                                        FB_Bacnet.StartStopCommand_142.bEnWrite := TRUE;
                                        FB_Bacnet.StartStopCommand_142.bVal := FALSE;
                                    16: 
                                        
                                        FB_Bacnet.StartStopCommand_143.bEnWrite := TRUE;
                                        FB_Bacnet.StartStopCommand_143.bVal := FALSE;
                                    17: 
                                        
                                        FB_Bacnet.StartStopCommand_144.bEnWrite := TRUE;
                                        FB_Bacnet.StartStopCommand_144.bVal := FALSE;
                                    18: 
                                        
                                        FB_Bacnet.StartStopCommand_145.bEnWrite := TRUE;
                                        FB_Bacnet.StartStopCommand_145.bVal := FALSE;
                                    19: 
                                        
                                        FB_Bacnet.StartStopCommand_146.bEnWrite := TRUE;
                                        FB_Bacnet.StartStopCommand_146.bVal := FALSE;
                                    20: 
                                        
                                        FB_Bacnet.StartStopCommand_147.bEnWrite := TRUE;
                                        FB_Bacnet.StartStopCommand_147.bVal := FALSE;
                                    21: 
                                        
                                        FB_Bacnet.StartStopCommand_148.bEnWrite := TRUE;
                                        FB_Bacnet.StartStopCommand_148.bVal := FALSE;
                                    22: 
                                        
                                        FB_Bacnet.StartStopCommand_176.bEnWrite := TRUE;
                                        FB_Bacnet.StartStopCommand_176.bVal := FALSE;
                                    23: 
                                        
                                        FB_Bacnet_b.StartStopCommand_241.bEnWrite := TRUE;
                                        FB_Bacnet_b.StartStopCommand_241.bVal := FALSE;
                                    24: 
                                        
                                        FB_Bacnet_b.StartStopCommand_227.bEnWrite := TRUE;
                                        FB_Bacnet_b.StartStopCommand_227.bVal := FALSE;
                                END_CASE
                            END_IF
                        END_FOR
                    END_IF
                END_IF
            END_IF

            // Weekend schedule
            IF currD = 0 OR currD = 6 THEN
                IF (wSchedWEHourStartF7_ <> wSchedWEHourEndF7_ OR wSchedWEMinStartF7_ <> wSchedWEMinEndF7_) THEN
                    // Schedule Unit ON
                    IF wSchedWEHourStartF7_ = currH AND wSchedWEMinStartF7_ = currM AND NOT bUnitTriggered THEN
                        bUnitTriggered := TRUE;
                        FOR i := 1 TO 24 DO
                            // Send command unit ON
                            IF bUnitF7_[i] THEN 
                                CASE i OF
                                    1: 
                                        
                                        FB_Bacnet.StartStopCommand_128.bEnWrite := TRUE;
                                        FB_Bacnet.StartStopCommand_128.bVal := TRUE;
                                    2: 
                                        
                                        FB_Bacnet.StartStopCommand_129.bEnWrite := TRUE;
                                        FB_Bacnet.StartStopCommand_129.bVal := TRUE;
                                    3: 
                                        
                                        FB_Bacnet.StartStopCommand_130.bEnWrite := TRUE;
                                        FB_Bacnet.StartStopCommand_130.bVal := TRUE;
                                    4: 
                                        
                                        FB_Bacnet.StartStopCommand_131.bEnWrite := TRUE;
                                        FB_Bacnet.StartStopCommand_131.bVal := TRUE;
                                    5: 
                                        
                                        FB_Bacnet.StartStopCommand_132.bEnWrite := TRUE;
                                        FB_Bacnet.StartStopCommand_132.bVal := TRUE;
                                    6: 
                                        
                                        FB_Bacnet.StartStopCommand_133.bEnWrite := TRUE;
                                        FB_Bacnet.StartStopCommand_133.bVal := TRUE;
                                    7: 
                                        
                                        FB_Bacnet.StartStopCommand_134.bEnWrite := TRUE;
                                        FB_Bacnet.StartStopCommand_134.bVal := TRUE;
                                    8: 
                                        
                                        FB_Bacnet.StartStopCommand_135.bEnWrite := TRUE;
                                        FB_Bacnet.StartStopCommand_135.bVal := TRUE;
                                    9: 
                                        
                                        FB_Bacnet.StartStopCommand_136.bEnWrite := TRUE;
                                        FB_Bacnet.StartStopCommand_136.bVal := TRUE;
                                    10: 
                                        
                                        FB_Bacnet.StartStopCommand_137.bEnWrite := TRUE;
                                        FB_Bacnet.StartStopCommand_137.bVal := TRUE;
                                    11: 
                                        
                                        FB_Bacnet.StartStopCommand_138.bEnWrite := TRUE;
                                        FB_Bacnet.StartStopCommand_138.bVal := TRUE;
                                    12: 
                                        
                                        FB_Bacnet.StartStopCommand_139.bEnWrite := TRUE;
                                        FB_Bacnet.StartStopCommand_139.bVal := TRUE;
                                    13: 
                                        
                                        FB_Bacnet.StartStopCommand_140.bEnWrite := TRUE;
                                        FB_Bacnet.StartStopCommand_140.bVal := TRUE;
                                    14: 
                                        
                                        FB_Bacnet.StartStopCommand_141.bEnWrite := TRUE;
                                        FB_Bacnet.StartStopCommand_141.bVal := TRUE;
                                    15: 
                                        
                                        FB_Bacnet.StartStopCommand_142.bEnWrite := TRUE;
                                        FB_Bacnet.StartStopCommand_142.bVal := TRUE;
                                    16: 
                                        
                                        FB_Bacnet.StartStopCommand_143.bEnWrite := TRUE;
                                        FB_Bacnet.StartStopCommand_143.bVal := TRUE;
                                    17: 
                                        
                                        FB_Bacnet.StartStopCommand_144.bEnWrite := TRUE;
                                        FB_Bacnet.StartStopCommand_144.bVal := TRUE;
                                    18: 
                                        
                                        FB_Bacnet.StartStopCommand_145.bEnWrite := TRUE;
                                        FB_Bacnet.StartStopCommand_145.bVal := TRUE;
                                    19: 
                                        
                                        FB_Bacnet.StartStopCommand_146.bEnWrite := TRUE;
                                        FB_Bacnet.StartStopCommand_146.bVal := TRUE;
                                    20: 
                                        
                                        FB_Bacnet.StartStopCommand_147.bEnWrite := TRUE;
                                        FB_Bacnet.StartStopCommand_147.bVal := TRUE;
                                    21: 
                                        
                                        FB_Bacnet.StartStopCommand_148.bEnWrite := TRUE;
                                        FB_Bacnet.StartStopCommand_148.bVal := TRUE;
                                    22: 
                                        
                                        FB_Bacnet.StartStopCommand_176.bEnWrite := TRUE;
                                        FB_Bacnet.StartStopCommand_176.bVal := TRUE;
                                    23: 
                                        
                                        FB_Bacnet_b.StartStopCommand_241.bEnWrite := TRUE;
                                        FB_Bacnet_b.StartStopCommand_241.bVal := TRUE;
                                    24: 
                                        
                                        FB_Bacnet_b.StartStopCommand_227.bEnWrite := TRUE;
                                        FB_Bacnet_b.StartStopCommand_227.bVal := TRUE;
                                END_CASE
                            END_IF
                        END_FOR
                    END_IF
                    // Schedule Unit OFF
                    IF wSchedWEHourEndF7_ = currH AND wSchedWEMinEndF7_ = currM AND NOT bUnitTriggered THEN
                        bUnitTriggered := TRUE;
                        FOR i := 1 TO 24 DO
                            // Send command unit OFF
                            IF bUnitF7_[i] THEN 
                                CASE i OF
                                    1: 
                                        
                                        FB_Bacnet.StartStopCommand_128.bEnWrite := TRUE;
                                        FB_Bacnet.StartStopCommand_128.bVal := FALSE;
                                    2: 
                                        
                                        FB_Bacnet.StartStopCommand_129.bEnWrite := TRUE;
                                        FB_Bacnet.StartStopCommand_129.bVal := FALSE;
                                    3: 
                                        
                                        FB_Bacnet.StartStopCommand_130.bEnWrite := TRUE;
                                        FB_Bacnet.StartStopCommand_130.bVal := FALSE;
                                    4: 
                                        
                                        FB_Bacnet.StartStopCommand_131.bEnWrite := TRUE;
                                        FB_Bacnet.StartStopCommand_131.bVal := FALSE;
                                    5: 
                                        
                                        FB_Bacnet.StartStopCommand_132.bEnWrite := TRUE;
                                        FB_Bacnet.StartStopCommand_132.bVal := FALSE;
                                    6: 
                                        
                                        FB_Bacnet.StartStopCommand_133.bEnWrite := TRUE;
                                        FB_Bacnet.StartStopCommand_133.bVal := FALSE;
                                    7: 
                                        
                                        FB_Bacnet.StartStopCommand_134.bEnWrite := TRUE;
                                        FB_Bacnet.StartStopCommand_134.bVal := FALSE;
                                    8: 
                                        
                                        FB_Bacnet.StartStopCommand_135.bEnWrite := TRUE;
                                        FB_Bacnet.StartStopCommand_135.bVal := FALSE;
                                    9: 
                                        
                                        FB_Bacnet.StartStopCommand_136.bEnWrite := TRUE;
                                        FB_Bacnet.StartStopCommand_136.bVal := FALSE;
                                    10: 
                                        
                                        FB_Bacnet.StartStopCommand_137.bEnWrite := TRUE;
                                        FB_Bacnet.StartStopCommand_137.bVal := FALSE;
                                    11: 
                                        
                                        FB_Bacnet.StartStopCommand_138.bEnWrite := TRUE;
                                        FB_Bacnet.StartStopCommand_138.bVal := FALSE;
                                    12: 
                                        
                                        FB_Bacnet.StartStopCommand_139.bEnWrite := TRUE;
                                        FB_Bacnet.StartStopCommand_139.bVal := FALSE;
                                    13: 
                                        
                                        FB_Bacnet.StartStopCommand_140.bEnWrite := TRUE;
                                        FB_Bacnet.StartStopCommand_140.bVal := FALSE;
                                    14: 
                                        
                                        FB_Bacnet.StartStopCommand_141.bEnWrite := TRUE;
                                        FB_Bacnet.StartStopCommand_141.bVal := FALSE;
                                    15: 
                                        
                                        FB_Bacnet.StartStopCommand_142.bEnWrite := TRUE;
                                        FB_Bacnet.StartStopCommand_142.bVal := FALSE;
                                    16: 
                                        
                                        FB_Bacnet.StartStopCommand_143.bEnWrite := TRUE;
                                        FB_Bacnet.StartStopCommand_143.bVal := FALSE;
                                    17: 
                                        
                                        FB_Bacnet.StartStopCommand_144.bEnWrite := TRUE;
                                        FB_Bacnet.StartStopCommand_144.bVal := FALSE;
                                    18: 
                                        
                                        FB_Bacnet.StartStopCommand_145.bEnWrite := TRUE;
                                        FB_Bacnet.StartStopCommand_145.bVal := FALSE;
                                    19: 
                                        
                                        FB_Bacnet.StartStopCommand_146.bEnWrite := TRUE;
                                        FB_Bacnet.StartStopCommand_146.bVal := FALSE;
                                    20: 
                                        
                                        FB_Bacnet.StartStopCommand_147.bEnWrite := TRUE;
                                        FB_Bacnet.StartStopCommand_147.bVal := FALSE;
                                    21: 
                                        
                                        FB_Bacnet.StartStopCommand_148.bEnWrite := TRUE;
                                        FB_Bacnet.StartStopCommand_148.bVal := FALSE;
                                    22: 
                                        
                                        FB_Bacnet.StartStopCommand_176.bEnWrite := TRUE;
                                        FB_Bacnet.StartStopCommand_176.bVal := FALSE;
                                    23: 
                                        
                                        FB_Bacnet_b.StartStopCommand_241.bEnWrite := TRUE;
                                        FB_Bacnet_b.StartStopCommand_241.bVal := FALSE;
                                    24: 
                                        
                                        FB_Bacnet_b.StartStopCommand_227.bEnWrite := TRUE;
                                        FB_Bacnet_b.StartStopCommand_227.bVal := FALSE;
                                END_CASE
                            END_IF
                        END_FOR
                    END_IF
                END_IF
            END_IF
        END_IF

END_FUNCTION_BLOCK

// ---- POUs/FB_Scheduler/FB_Scheduler_F8.TcPOU

      FUNCTION_BLOCK FB_Scheduler_F8
      VAR_INPUT
          currH : WORD;
          currM : WORD;
          currD : WORD;
      END_VAR
      VAR_IN_OUT
          FB_Bacnet : FB_BACnet_DAIKIN_MasterStation_III_No_2;
      END_VAR
      VAR
          i : INT;
          bUnitTriggered : BOOL := FALSE; // Flag to track execution
          prevMinute : WORD := 0;        // Track previous minute
      END_VAR
      VAR PERSISTENT
          // Scheduler variables
          bEnSchedF8_ : BOOL := FALSE;
          wSchedWDHourStartF8_, wSchedWDMinStartF8_ : WORD;
          wSchedWEHourStartF8_, wSchedWEMinStartF8_ : WORD;
          wSchedWDHourEndF8_, wSchedWDMinEndF8_ : WORD;
          wSchedWEHourEndF8_, wSchedWEMinEndF8_ : WORD;
          // Unit variables
          bUnitF8_ : ARRAY [1..22] OF BOOL;
      END_VAR


        // Reset trigger flag at minute change or at the exact scheduled time
        IF currM <> prevMinute OR 
           (currH = wSchedWDHourStartF8_ AND currM = wSchedWDMinStartF8_) OR 
           (currH = wSchedWDHourEndF8_ AND currM = wSchedWDMinEndF8_) THEN
            bUnitTriggered := FALSE;
            prevMinute := currM;
        END_IF

        // Unit Schedule Enable
        IF bEnSchedF8_ THEN
            // Weekday schedule
            IF currD >= 1 AND currD <= 5 THEN
                IF (wSchedWDHourStartF8_ <> wSchedWDHourEndF8_ OR wSchedWDMinStartF8_ <> wSchedWDMinEndF8_) THEN
                    // Schedule Unit ON
                    IF wSchedWDHourStartF8_ = currH AND wSchedWDMinStartF8_ = currM AND NOT bUnitTriggered THEN
                        bUnitTriggered := TRUE;
                        FOR i := 1 TO 22 DO
                            // Send command unit ON
                            IF bUnitF8_[i] THEN 
                                CASE i OF
                                    1: 
                                        FB_Bacnet.StartStopCommand_192.bEnWrite := TRUE;
                                        FB_Bacnet.StartStopCommand_192.bVal := TRUE;
                                    2: 
                                        FB_Bacnet.StartStopCommand_193.bEnWrite := TRUE;
                                        FB_Bacnet.StartStopCommand_193.bVal := TRUE;
                                    3: 
                                        FB_Bacnet.StartStopCommand_194.bEnWrite := TRUE;
                                        FB_Bacnet.StartStopCommand_194.bVal := TRUE;
                                    4: 
                                        FB_Bacnet.StartStopCommand_195.bEnWrite := TRUE;
                                        FB_Bacnet.StartStopCommand_195.bVal := TRUE;
                                    5: 
                                        FB_Bacnet.StartStopCommand_196.bEnWrite := TRUE;
                                        FB_Bacnet.StartStopCommand_196.bVal := TRUE;
                                    6: 
                                        FB_Bacnet.StartStopCommand_197.bEnWrite := TRUE;
                                        FB_Bacnet.StartStopCommand_197.bVal := TRUE;
                                    7: 
                                        FB_Bacnet.StartStopCommand_198.bEnWrite := TRUE;
                                        FB_Bacnet.StartStopCommand_198.bVal := TRUE;
                                    8: 
                                        FB_Bacnet.StartStopCommand_199.bEnWrite := TRUE;
                                        FB_Bacnet.StartStopCommand_199.bVal := TRUE;
                                    9: 
                                        FB_Bacnet.StartStopCommand_200.bEnWrite := TRUE;
                                        FB_Bacnet.StartStopCommand_200.bVal := TRUE;
                                    10: 
                                        FB_Bacnet.StartStopCommand_201.bEnWrite := TRUE;
                                        FB_Bacnet.StartStopCommand_201.bVal := TRUE;
                                    11: 
                                        FB_Bacnet.StartStopCommand_202.bEnWrite := TRUE;
                                        FB_Bacnet.StartStopCommand_202.bVal := TRUE;
                                    12: 
                                        FB_Bacnet.StartStopCommand_203.bEnWrite := TRUE;
                                        FB_Bacnet.StartStopCommand_203.bVal := TRUE;
                                    13: 
                                        FB_Bacnet.StartStopCommand_204.bEnWrite := TRUE;
                                        FB_Bacnet.StartStopCommand_204.bVal := TRUE;
                                    14: 
                                        FB_Bacnet.StartStopCommand_205.bEnWrite := TRUE;
                                        FB_Bacnet.StartStopCommand_205.bVal := TRUE;
                                    15: 
                                        FB_Bacnet.StartStopCommand_206.bEnWrite := TRUE;
                                        FB_Bacnet.StartStopCommand_206.bVal := TRUE;
                                    16: 
                                        FB_Bacnet.StartStopCommand_207.bEnWrite := TRUE;
                                        FB_Bacnet.StartStopCommand_207.bVal := TRUE;
                                    17: 
                                        FB_Bacnet.StartStopCommand_208.bEnWrite := TRUE;
                                        FB_Bacnet.StartStopCommand_208.bVal := TRUE;
                                    18: 
                                        FB_Bacnet.StartStopCommand_209.bEnWrite := TRUE;
                                        FB_Bacnet.StartStopCommand_209.bVal := TRUE;
                                    19: 
                                        FB_Bacnet.StartStopCommand_210.bEnWrite := TRUE;
                                        FB_Bacnet.StartStopCommand_210.bVal := TRUE;
                                    20: 
                                        FB_Bacnet.StartStopCommand_211.bEnWrite := TRUE;
                                        FB_Bacnet.StartStopCommand_211.bVal := TRUE;
                                    21: 
                                        FB_Bacnet.StartStopCommand_212.bEnWrite := TRUE;
                                        FB_Bacnet.StartStopCommand_212.bVal := TRUE;
                                    22: 
                                        FB_Bacnet.StartStopCommand_224.bEnWrite := TRUE;
                                        FB_Bacnet.StartStopCommand_224.bVal := TRUE;
                                END_CASE
                            END_IF
                        END_FOR
                    END_IF
                    // Schedule Unit OFF
                    IF wSchedWDHourEndF8_ = currH AND wSchedWDMinEndF8_ = currM AND NOT bUnitTriggered THEN
                        bUnitTriggered := TRUE;
                        FOR i := 1 TO 22 DO
                            // Send command unit OFF
                            IF bUnitF8_[i] THEN 
                                CASE i OF
                                    1: 
                                        FB_Bacnet.StartStopCommand_192.bEnWrite := TRUE;
                                        FB_Bacnet.StartStopCommand_192.bVal := FALSE;
                                    2: 
                                        FB_Bacnet.StartStopCommand_193.bEnWrite := TRUE;
                                        FB_Bacnet.StartStopCommand_193.bVal := FALSE;
                                    3: 
                                        FB_Bacnet.StartStopCommand_194.bEnWrite := TRUE;
                                        FB_Bacnet.StartStopCommand_194.bVal := FALSE;
                                    4: 
                                        FB_Bacnet.StartStopCommand_195.bEnWrite := TRUE;
                                        FB_Bacnet.StartStopCommand_195.bVal := FALSE;
                                    5: 
                                        FB_Bacnet.StartStopCommand_196.bEnWrite := TRUE;
                                        FB_Bacnet.StartStopCommand_196.bVal := FALSE;
                                    6: 
                                        FB_Bacnet.StartStopCommand_197.bEnWrite := TRUE;
                                        FB_Bacnet.StartStopCommand_197.bVal := FALSE;
                                    7: 
                                        FB_Bacnet.StartStopCommand_198.bEnWrite := TRUE;
                                        FB_Bacnet.StartStopCommand_198.bVal := FALSE;
                                    8: 
                                        FB_Bacnet.StartStopCommand_199.bEnWrite := TRUE;
                                        FB_Bacnet.StartStopCommand_199.bVal := FALSE;
                                    9: 
                                        FB_Bacnet.StartStopCommand_200.bEnWrite := TRUE;
                                        FB_Bacnet.StartStopCommand_200.bVal := FALSE;
                                    10: 
                                        FB_Bacnet.StartStopCommand_201.bEnWrite := TRUE;
                                        FB_Bacnet.StartStopCommand_201.bVal := FALSE;
                                    11: 
                                        FB_Bacnet.StartStopCommand_202.bEnWrite := TRUE;
                                        FB_Bacnet.StartStopCommand_202.bVal := FALSE;
                                    12: 
                                        FB_Bacnet.StartStopCommand_203.bEnWrite := TRUE;
                                        FB_Bacnet.StartStopCommand_203.bVal := FALSE;
                                    13: 
                                        FB_Bacnet.StartStopCommand_204.bEnWrite := TRUE;
                                        FB_Bacnet.StartStopCommand_204.bVal := FALSE;
                                    14: 
                                        FB_Bacnet.StartStopCommand_205.bEnWrite := TRUE;
                                        FB_Bacnet.StartStopCommand_205.bVal := FALSE;
                                    15: 
                                        FB_Bacnet.StartStopCommand_206.bEnWrite := TRUE;
                                        FB_Bacnet.StartStopCommand_206.bVal := FALSE;
                                    16: 
                                        FB_Bacnet.StartStopCommand_207.bEnWrite := TRUE;
                                        FB_Bacnet.StartStopCommand_207.bVal := FALSE;
                                    17: 
                                        FB_Bacnet.StartStopCommand_208.bEnWrite := TRUE;
                                        FB_Bacnet.StartStopCommand_208.bVal := FALSE;
                                    18: 
                                        FB_Bacnet.StartStopCommand_209.bEnWrite := TRUE;
                                        FB_Bacnet.StartStopCommand_209.bVal := FALSE;
                                    19: 
                                        FB_Bacnet.StartStopCommand_210.bEnWrite := TRUE;
                                        FB_Bacnet.StartStopCommand_210.bVal := FALSE;
                                    20: 
                                        FB_Bacnet.StartStopCommand_211.bEnWrite := TRUE;
                                        FB_Bacnet.StartStopCommand_211.bVal := FALSE;
                                    21: 
                                        FB_Bacnet.StartStopCommand_212.bEnWrite := TRUE;
                                        FB_Bacnet.StartStopCommand_212.bVal := FALSE;
                                    22: 
                                        FB_Bacnet.StartStopCommand_224.bEnWrite := TRUE;
                                        FB_Bacnet.StartStopCommand_224.bVal := FALSE;
                                END_CASE
                            END_IF
                        END_FOR
                    END_IF
                END_IF
            END_IF

            // Weekend schedule
            IF currD = 0 OR currD = 6 THEN
                IF (wSchedWEHourStartF8_ <> wSchedWEHourEndF8_ OR wSchedWEMinStartF8_ <> wSchedWEMinEndF8_) THEN
                    // Schedule Unit ON
                    IF wSchedWEHourStartF8_ = currH AND wSchedWEMinStartF8_ = currM AND NOT bUnitTriggered THEN
                        bUnitTriggered := TRUE;
                        FOR i := 1 TO 22 DO
                            // Send command unit ON
                            IF bUnitF8_[i] THEN 
                                CASE i OF
                                    1: 
                                        FB_Bacnet.StartStopCommand_192.bEnWrite := TRUE;
                                        FB_Bacnet.StartStopCommand_192.bVal := TRUE;
                                    2: 
                                        FB_Bacnet.StartStopCommand_193.bEnWrite := TRUE;
                                        FB_Bacnet.StartStopCommand_193.bVal := TRUE;
                                    3: 
                                        FB_Bacnet.StartStopCommand_194.bEnWrite := TRUE;
                                        FB_Bacnet.StartStopCommand_194.bVal := TRUE;
                                    4: 
                                        FB_Bacnet.StartStopCommand_195.bEnWrite := TRUE;
                                        FB_Bacnet.StartStopCommand_195.bVal := TRUE;
                                    5: 
                                        FB_Bacnet.StartStopCommand_196.bEnWrite := TRUE;
                                        FB_Bacnet.StartStopCommand_196.bVal := TRUE;
                                    6: 
                                        FB_Bacnet.StartStopCommand_197.bEnWrite := TRUE;
                                        FB_Bacnet.StartStopCommand_197.bVal := TRUE;
                                    7: 
                                        FB_Bacnet.StartStopCommand_198.bEnWrite := TRUE;
                                        FB_Bacnet.StartStopCommand_198.bVal := TRUE;
                                    8: 
                                        FB_Bacnet.StartStopCommand_199.bEnWrite := TRUE;
                                        FB_Bacnet.StartStopCommand_199.bVal := TRUE;
                                    9: 
                                        FB_Bacnet.StartStopCommand_200.bEnWrite := TRUE;
                                        FB_Bacnet.StartStopCommand_200.bVal := TRUE;
                                    10: 
                                        FB_Bacnet.StartStopCommand_201.bEnWrite := TRUE;
                                        FB_Bacnet.StartStopCommand_201.bVal := TRUE;
                                    11: 
                                        FB_Bacnet.StartStopCommand_202.bEnWrite := TRUE;
                                        FB_Bacnet.StartStopCommand_202.bVal := TRUE;
                                    12: 
                                        FB_Bacnet.StartStopCommand_203.bEnWrite := TRUE;
                                        FB_Bacnet.StartStopCommand_203.bVal := TRUE;
                                    13: 
                                        FB_Bacnet.StartStopCommand_204.bEnWrite := TRUE;
                                        FB_Bacnet.StartStopCommand_204.bVal := TRUE;
                                    14: 
                                        FB_Bacnet.StartStopCommand_205.bEnWrite := TRUE;
                                        FB_Bacnet.StartStopCommand_205.bVal := TRUE;
                                    15: 
                                        FB_Bacnet.StartStopCommand_206.bEnWrite := TRUE;
                                        FB_Bacnet.StartStopCommand_206.bVal := TRUE;
                                    16: 
                                        FB_Bacnet.StartStopCommand_207.bEnWrite := TRUE;
                                        FB_Bacnet.StartStopCommand_207.bVal := TRUE;
                                    17: 
                                        FB_Bacnet.StartStopCommand_208.bEnWrite := TRUE;
                                        FB_Bacnet.StartStopCommand_208.bVal := TRUE;
                                    18: 
                                        FB_Bacnet.StartStopCommand_209.bEnWrite := TRUE;
                                        FB_Bacnet.StartStopCommand_209.bVal := TRUE;
                                    19: 
                                        FB_Bacnet.StartStopCommand_210.bEnWrite := TRUE;
                                        FB_Bacnet.StartStopCommand_210.bVal := TRUE;
                                    20: 
                                        FB_Bacnet.StartStopCommand_211.bEnWrite := TRUE;
                                        FB_Bacnet.StartStopCommand_211.bVal := TRUE;
                                    21: 
                                        FB_Bacnet.StartStopCommand_212.bEnWrite := TRUE;
                                        FB_Bacnet.StartStopCommand_212.bVal := TRUE;
                                    22: 
                                        FB_Bacnet.StartStopCommand_224.bEnWrite := TRUE;
                                        FB_Bacnet.StartStopCommand_224.bVal := TRUE;
                                END_CASE
                            END_IF
                        END_FOR
                    END_IF
                    // Schedule Unit OFF
                    IF wSchedWEHourEndF8_ = currH AND wSchedWEMinEndF8_ = currM AND NOT bUnitTriggered THEN
                        bUnitTriggered := TRUE;
                        FOR i := 1 TO 22 DO
                            // Send command unit OFF
                            IF bUnitF8_[i] THEN 
                                CASE i OF
                                    1: 
                                        FB_Bacnet.StartStopCommand_192.bEnWrite := TRUE;
                                        FB_Bacnet.StartStopCommand_192.bVal := FALSE;
                                    2: 
                                        FB_Bacnet.StartStopCommand_193.bEnWrite := TRUE;
                                        FB_Bacnet.StartStopCommand_193.bVal := FALSE;
                                    3: 
                                        FB_Bacnet.StartStopCommand_194.bEnWrite := TRUE;
                                        FB_Bacnet.StartStopCommand_194.bVal := FALSE;
                                    4: 
                                        FB_Bacnet.StartStopCommand_195.bEnWrite := TRUE;
                                        FB_Bacnet.StartStopCommand_195.bVal := FALSE;
                                    5: 
                                        FB_Bacnet.StartStopCommand_196.bEnWrite := TRUE;
                                        FB_Bacnet.StartStopCommand_196.bVal := FALSE;
                                    6: 
                                        FB_Bacnet.StartStopCommand_197.bEnWrite := TRUE;
                                        FB_Bacnet.StartStopCommand_197.bVal := FALSE;
                                    7: 
                                        FB_Bacnet.StartStopCommand_198.bEnWrite := TRUE;
                                        FB_Bacnet.StartStopCommand_198.bVal := FALSE;
                                    8: 
                                        FB_Bacnet.StartStopCommand_199.bEnWrite := TRUE;
                                        FB_Bacnet.StartStopCommand_199.bVal := FALSE;
                                    9: 
                                        FB_Bacnet.StartStopCommand_200.bEnWrite := TRUE;
                                        FB_Bacnet.StartStopCommand_200.bVal := FALSE;
                                    10: 
                                        FB_Bacnet.StartStopCommand_201.bEnWrite := TRUE;
                                        FB_Bacnet.StartStopCommand_201.bVal := FALSE;
                                    11: 
                                        FB_Bacnet.StartStopCommand_202.bEnWrite := TRUE;
                                        FB_Bacnet.StartStopCommand_202.bVal := FALSE;
                                    12: 
                                        FB_Bacnet.StartStopCommand_203.bEnWrite := TRUE;
                                        FB_Bacnet.StartStopCommand_203.bVal := FALSE;
                                    13: 
                                        FB_Bacnet.StartStopCommand_204.bEnWrite := TRUE;
                                        FB_Bacnet.StartStopCommand_204.bVal := FALSE;
                                    14: 
                                        FB_Bacnet.StartStopCommand_205.bEnWrite := TRUE;
                                        FB_Bacnet.StartStopCommand_205.bVal := FALSE;
                                    15: 
                                        FB_Bacnet.StartStopCommand_206.bEnWrite := TRUE;
                                        FB_Bacnet.StartStopCommand_206.bVal := FALSE;
                                    16: 
                                        FB_Bacnet.StartStopCommand_207.bEnWrite := TRUE;
                                        FB_Bacnet.StartStopCommand_207.bVal := FALSE;
                                    17: 
                                        FB_Bacnet.StartStopCommand_208.bEnWrite := TRUE;
                                        FB_Bacnet.StartStopCommand_208.bVal := FALSE;
                                    18: 
                                        FB_Bacnet.StartStopCommand_209.bEnWrite := TRUE;
                                        FB_Bacnet.StartStopCommand_209.bVal := FALSE;
                                    19: 
                                        FB_Bacnet.StartStopCommand_210.bEnWrite := TRUE;
                                        FB_Bacnet.StartStopCommand_210.bVal := FALSE;
                                    20: 
                                        FB_Bacnet.StartStopCommand_211.bEnWrite := TRUE;
                                        FB_Bacnet.StartStopCommand_211.bVal := FALSE;
                                    21: 
                                        FB_Bacnet.StartStopCommand_212.bEnWrite := TRUE;
                                        FB_Bacnet.StartStopCommand_212.bVal := FALSE;
                                    22: 
                                        FB_Bacnet.StartStopCommand_224.bEnWrite := TRUE;
                                        FB_Bacnet.StartStopCommand_224.bVal := FALSE;
                                END_CASE
                            END_IF
                        END_FOR
                    END_IF
                END_IF
            END_IF
        END_IF

END_FUNCTION_BLOCK

// ---- POUs/FB_Scheduler/FB_Scheduler_F9.TcPOU

      FUNCTION_BLOCK FB_Scheduler_F9
      VAR_INPUT
          currH : WORD;
          currM : WORD;
          currD : WORD;
      END_VAR
      VAR_IN_OUT
          FB_Bacnet : FB_BACnet_DAIKIN_MasterStation_III_No_3;
          FB_Bacnet_b : FB_BACnet_DAIKIN_MasterStation_III_No_2;
      END_VAR
      VAR
          i : INT;
          bUnitTriggered : BOOL := FALSE; // Flag to track execution
          prevMinute : WORD := 0;        // Track previous minute
      END_VAR
      VAR PERSISTENT
          // Scheduler variables
          bEnSchedF9_ : BOOL := FALSE;
          wSchedWDHourStartF9_, wSchedWDMinStartF9_ : WORD;
          wSchedWEHourStartF9_, wSchedWEMinStartF9_ : WORD;
          wSchedWDHourEndF9_, wSchedWDMinEndF9_ : WORD;
          wSchedWEHourEndF9_, wSchedWEMinEndF9_ : WORD;
          // Unit variables
          bUnitF9_ : ARRAY [1..22] OF BOOL;
      END_VAR


        // Reset trigger flag at minute change or at the exact scheduled time
        IF currM <> prevMinute OR 
           (currH = wSchedWDHourStartF9_ AND currM = wSchedWDMinStartF9_) OR 
           (currH = wSchedWDHourEndF9_ AND currM = wSchedWDMinEndF9_) THEN
            bUnitTriggered := FALSE;
            prevMinute := currM;
        END_IF

        // Unit Schedule Enable
        IF bEnSchedF9_ THEN
            // Weekday schedule
            IF currD >= 1 AND currD <= 5 THEN
                IF (wSchedWDHourStartF9_ <> wSchedWDHourEndF9_ OR wSchedWDMinStartF9_ <> wSchedWDMinEndF9_) THEN
                    // Schedule Unit ON
                    IF wSchedWDHourStartF9_ = currH AND wSchedWDMinStartF9_ = currM AND NOT bUnitTriggered THEN
                        bUnitTriggered := TRUE;
                        FOR i := 1 TO 22 DO
                            // Send command unit ON
                            IF bUnitF9_[i] THEN 
                                CASE i OF
                                    1: 
                                        
                                        FB_Bacnet.StartStopCommand_000.bEnWrite := TRUE;
                                        FB_Bacnet.StartStopCommand_000.bVal := TRUE;
                                    2: 
                                        
                                        FB_Bacnet.StartStopCommand_001.bEnWrite := TRUE;
                                        FB_Bacnet.StartStopCommand_001.bVal := TRUE;
                                    3: 
                                        
                                        FB_Bacnet.StartStopCommand_002.bEnWrite := TRUE;
                                        FB_Bacnet.StartStopCommand_002.bVal := TRUE;
                                    4: 
                                        
                                        FB_Bacnet.StartStopCommand_003.bEnWrite := TRUE;
                                        FB_Bacnet.StartStopCommand_003.bVal := TRUE;
                                    5: 
                                        
                                        FB_Bacnet.StartStopCommand_004.bEnWrite := TRUE;
                                        FB_Bacnet.StartStopCommand_004.bVal := TRUE;
                                    6: 
                                        
                                        FB_Bacnet.StartStopCommand_005.bEnWrite := TRUE;
                                        FB_Bacnet.StartStopCommand_005.bVal := TRUE;
                                    7: 
                                        
                                        FB_Bacnet.StartStopCommand_006.bEnWrite := TRUE;
                                        FB_Bacnet.StartStopCommand_006.bVal := TRUE;
                                    8: 
                                        
                                        FB_Bacnet.StartStopCommand_007.bEnWrite := TRUE;
                                        FB_Bacnet.StartStopCommand_007.bVal := TRUE;
                                    9: 
                                        
                                        FB_Bacnet.StartStopCommand_008.bEnWrite := TRUE;
                                        FB_Bacnet.StartStopCommand_008.bVal := TRUE;
                                    10: 
                                        
                                        FB_Bacnet.StartStopCommand_009.bEnWrite := TRUE;
                                        FB_Bacnet.StartStopCommand_009.bVal := TRUE;
                                    11: 
                                        
                                        FB_Bacnet.StartStopCommand_010.bEnWrite := TRUE;
                                        FB_Bacnet.StartStopCommand_010.bVal := TRUE;
                                    12: 
                                        
                                        FB_Bacnet.StartStopCommand_011.bEnWrite := TRUE;
                                        FB_Bacnet.StartStopCommand_011.bVal := TRUE;
                                    13: 
                                        
                                        FB_Bacnet.StartStopCommand_012.bEnWrite := TRUE;
                                        FB_Bacnet.StartStopCommand_012.bVal := TRUE;
                                    14: 
                                        
                                        FB_Bacnet.StartStopCommand_013.bEnWrite := TRUE;
                                        FB_Bacnet.StartStopCommand_013.bVal := TRUE;
                                    15: 
                                        
                                        FB_Bacnet.StartStopCommand_014.bEnWrite := TRUE;
                                        FB_Bacnet.StartStopCommand_014.bVal := TRUE;
                                    16: 
                                        
                                        FB_Bacnet.StartStopCommand_015.bEnWrite := TRUE;
                                        FB_Bacnet.StartStopCommand_015.bVal := TRUE;
                                    17: 
                                        
                                        FB_Bacnet.StartStopCommand_016.bEnWrite := TRUE;
                                        FB_Bacnet.StartStopCommand_016.bVal := TRUE;
                                    18: 
                                        
                                        FB_Bacnet.StartStopCommand_017.bEnWrite := TRUE;
                                        FB_Bacnet.StartStopCommand_017.bVal := TRUE;
                                    19: 
                                        
                                        FB_Bacnet.StartStopCommand_018.bEnWrite := TRUE;
                                        FB_Bacnet.StartStopCommand_018.bVal := TRUE;
                                    20: 
                                        
                                        FB_Bacnet.StartStopCommand_019.bEnWrite := TRUE;
                                        FB_Bacnet.StartStopCommand_019.bVal := TRUE;
                                    21: 
                                        
                                        FB_Bacnet.StartStopCommand_020.bEnWrite := TRUE;
                                        FB_Bacnet.StartStopCommand_020.bVal := TRUE;
                                    22: 
                                        
                                        FB_Bacnet_b.StartStopCommand_225.bEnWrite := TRUE;
                                        FB_Bacnet_b.StartStopCommand_225.bVal := TRUE;
                                END_CASE
                            END_IF
                        END_FOR
                    END_IF
                    // Schedule Unit OFF
                    IF wSchedWDHourEndF9_ = currH AND wSchedWDMinEndF9_ = currM AND NOT bUnitTriggered THEN
                        bUnitTriggered := TRUE;
                        FOR i := 1 TO 22 DO
                            // Send command unit OFF
                            IF bUnitF9_[i] THEN 
                                CASE i OF
                                    1: 
                                        
                                        FB_Bacnet.StartStopCommand_000.bEnWrite := TRUE;
                                        FB_Bacnet.StartStopCommand_000.bVal := FALSE;
                                    2: 
                                        
                                        FB_Bacnet.StartStopCommand_001.bEnWrite := TRUE;
                                        FB_Bacnet.StartStopCommand_001.bVal := FALSE;
                                    3: 
                                        
                                        FB_Bacnet.StartStopCommand_002.bEnWrite := TRUE;
                                        FB_Bacnet.StartStopCommand_002.bVal := FALSE;
                                    4: 
                                        
                                        FB_Bacnet.StartStopCommand_003.bEnWrite := TRUE;
                                        FB_Bacnet.StartStopCommand_003.bVal := FALSE;
                                    5: 
                                        
                                        FB_Bacnet.StartStopCommand_004.bEnWrite := TRUE;
                                        FB_Bacnet.StartStopCommand_004.bVal := FALSE;
                                    6: 
                                        
                                        FB_Bacnet.StartStopCommand_005.bEnWrite := TRUE;
                                        FB_Bacnet.StartStopCommand_005.bVal := FALSE;
                                    7: 
                                        
                                        FB_Bacnet.StartStopCommand_006.bEnWrite := TRUE;
                                        FB_Bacnet.StartStopCommand_006.bVal := FALSE;
                                    8: 
                                        
                                        FB_Bacnet.StartStopCommand_007.bEnWrite := TRUE;
                                        FB_Bacnet.StartStopCommand_007.bVal := FALSE;
                                    9: 
                                        
                                        FB_Bacnet.StartStopCommand_008.bEnWrite := TRUE;
                                        FB_Bacnet.StartStopCommand_008.bVal := FALSE;
                                    10: 
                                        
                                        FB_Bacnet.StartStopCommand_009.bEnWrite := TRUE;
                                        FB_Bacnet.StartStopCommand_009.bVal := FALSE;
                                    11: 
                                        
                                        FB_Bacnet.StartStopCommand_010.bEnWrite := TRUE;
                                        FB_Bacnet.StartStopCommand_010.bVal := FALSE;
                                    12: 
                                        
                                        FB_Bacnet.StartStopCommand_011.bEnWrite := TRUE;
                                        FB_Bacnet.StartStopCommand_011.bVal := FALSE;
                                    13: 
                                        
                                        FB_Bacnet.StartStopCommand_012.bEnWrite := TRUE;
                                        FB_Bacnet.StartStopCommand_012.bVal := FALSE;
                                    14: 
                                        
                                        FB_Bacnet.StartStopCommand_013.bEnWrite := TRUE;
                                        FB_Bacnet.StartStopCommand_013.bVal := FALSE;
                                    15: 
                                        
                                        FB_Bacnet.StartStopCommand_014.bEnWrite := TRUE;
                                        FB_Bacnet.StartStopCommand_014.bVal := FALSE;
                                    16: 
                                        
                                        FB_Bacnet.StartStopCommand_015.bEnWrite := TRUE;
                                        FB_Bacnet.StartStopCommand_015.bVal := FALSE;
                                    17: 
                                        
                                        FB_Bacnet.StartStopCommand_016.bEnWrite := TRUE;
                                        FB_Bacnet.StartStopCommand_016.bVal := FALSE;
                                    18: 
                                        
                                        FB_Bacnet.StartStopCommand_017.bEnWrite := TRUE;
                                        FB_Bacnet.StartStopCommand_017.bVal := FALSE;
                                    19: 
                                        
                                        FB_Bacnet.StartStopCommand_018.bEnWrite := TRUE;
                                        FB_Bacnet.StartStopCommand_018.bVal := FALSE;
                                    20: 
                                        
                                        FB_Bacnet.StartStopCommand_019.bEnWrite := TRUE;
                                        FB_Bacnet.StartStopCommand_019.bVal := FALSE;
                                    21: 
                                        
                                        FB_Bacnet.StartStopCommand_020.bEnWrite := TRUE;
                                        FB_Bacnet.StartStopCommand_020.bVal := FALSE;
                                    22: 
                                        
                                        FB_Bacnet_b.StartStopCommand_225.bEnWrite := TRUE;
                                        FB_Bacnet_b.StartStopCommand_225.bVal := FALSE;
                                END_CASE
                            END_IF
                        END_FOR
                    END_IF
                END_IF
            END_IF

            // Weekend schedule
            IF currD = 0 OR currD = 6 THEN
                IF (wSchedWEHourStartF9_ <> wSchedWEHourEndF9_ OR wSchedWEMinStartF9_ <> wSchedWEMinEndF9_) THEN
                    // Schedule Unit ON
                    IF wSchedWEHourStartF9_ = currH AND wSchedWEMinStartF9_ = currM AND NOT bUnitTriggered THEN
                        bUnitTriggered := TRUE;
                        FOR i := 1 TO 22 DO
                            // Send command unit ON
                            IF bUnitF9_[i] THEN 
                                CASE i OF
                                    1: 
                                        
                                        FB_Bacnet.StartStopCommand_000.bEnWrite := TRUE;
                                        FB_Bacnet.StartStopCommand_000.bVal := TRUE;
                                    2: 
                                        
                                        FB_Bacnet.StartStopCommand_001.bEnWrite := TRUE;
                                        FB_Bacnet.StartStopCommand_001.bVal := TRUE;
                                    3: 
                                        
                                        FB_Bacnet.StartStopCommand_002.bEnWrite := TRUE;
                                        FB_Bacnet.StartStopCommand_002.bVal := TRUE;
                                    4: 
                                        
                                        FB_Bacnet.StartStopCommand_003.bEnWrite := TRUE;
                                        FB_Bacnet.StartStopCommand_003.bVal := TRUE;
                                    5: 
                                        
                                        FB_Bacnet.StartStopCommand_004.bEnWrite := TRUE;
                                        FB_Bacnet.StartStopCommand_004.bVal := TRUE;
                                    6: 
                                        
                                        FB_Bacnet.StartStopCommand_005.bEnWrite := TRUE;
                                        FB_Bacnet.StartStopCommand_005.bVal := TRUE;
                                    7: 
                                        
                                        FB_Bacnet.StartStopCommand_006.bEnWrite := TRUE;
                                        FB_Bacnet.StartStopCommand_006.bVal := TRUE;
                                    8: 
                                        
                                        FB_Bacnet.StartStopCommand_007.bEnWrite := TRUE;
                                        FB_Bacnet.StartStopCommand_007.bVal := TRUE;
                                    9: 
                                        
                                        FB_Bacnet.StartStopCommand_008.bEnWrite := TRUE;
                                        FB_Bacnet.StartStopCommand_008.bVal := TRUE;
                                    10: 
                                        
                                        FB_Bacnet.StartStopCommand_009.bEnWrite := TRUE;
                                        FB_Bacnet.StartStopCommand_009.bVal := TRUE;
                                    11: 
                                        
                                        FB_Bacnet.StartStopCommand_010.bEnWrite := TRUE;
                                        FB_Bacnet.StartStopCommand_010.bVal := TRUE;
                                    12: 
                                        
                                        FB_Bacnet.StartStopCommand_011.bEnWrite := TRUE;
                                        FB_Bacnet.StartStopCommand_011.bVal := TRUE;
                                    13: 
                                        
                                        FB_Bacnet.StartStopCommand_012.bEnWrite := TRUE;
                                        FB_Bacnet.StartStopCommand_012.bVal := TRUE;
                                    14: 
                                        
                                        FB_Bacnet.StartStopCommand_013.bEnWrite := TRUE;
                                        FB_Bacnet.StartStopCommand_013.bVal := TRUE;
                                    15: 
                                        
                                        FB_Bacnet.StartStopCommand_014.bEnWrite := TRUE;
                                        FB_Bacnet.StartStopCommand_014.bVal := TRUE;
                                    16: 
                                        
                                        FB_Bacnet.StartStopCommand_015.bEnWrite := TRUE;
                                        FB_Bacnet.StartStopCommand_015.bVal := TRUE;
                                    17: 
                                        
                                        FB_Bacnet.StartStopCommand_016.bEnWrite := TRUE;
                                        FB_Bacnet.StartStopCommand_016.bVal := TRUE;
                                    18: 
                                        
                                        FB_Bacnet.StartStopCommand_017.bEnWrite := TRUE;
                                        FB_Bacnet.StartStopCommand_017.bVal := TRUE;
                                    19: 
                                        
                                        FB_Bacnet.StartStopCommand_018.bEnWrite := TRUE;
                                        FB_Bacnet.StartStopCommand_018.bVal := TRUE;
                                    20: 
                                        
                                        FB_Bacnet.StartStopCommand_019.bEnWrite := TRUE;
                                        FB_Bacnet.StartStopCommand_019.bVal := TRUE;
                                    21: 
                                        
                                        FB_Bacnet.StartStopCommand_020.bEnWrite := TRUE;
                                        FB_Bacnet.StartStopCommand_020.bVal := TRUE;
                                    22: 
                                        
                                        FB_Bacnet_b.StartStopCommand_225.bEnWrite := TRUE;
                                        FB_Bacnet_b.StartStopCommand_225.bVal := TRUE;
                                END_CASE
                            END_IF
                        END_FOR
                    END_IF
                    // Schedule Unit OFF
                    IF wSchedWEHourEndF9_ = currH AND wSchedWEMinEndF9_ = currM AND NOT bUnitTriggered THEN
                        bUnitTriggered := TRUE;
                        FOR i := 1 TO 22 DO
                            // Send command unit OFF
                            IF bUnitF9_[i] THEN 
                                CASE i OF
                                    1: 
                                        
                                        FB_Bacnet.StartStopCommand_000.bEnWrite := TRUE;
                                        FB_Bacnet.StartStopCommand_000.bVal := FALSE;
                                    2: 
                                        
                                        FB_Bacnet.StartStopCommand_001.bEnWrite := TRUE;
                                        FB_Bacnet.StartStopCommand_001.bVal := FALSE;
                                    3: 
                                        
                                        FB_Bacnet.StartStopCommand_002.bEnWrite := TRUE;
                                        FB_Bacnet.StartStopCommand_002.bVal := FALSE;
                                    4: 
                                        
                                        FB_Bacnet.StartStopCommand_003.bEnWrite := TRUE;
                                        FB_Bacnet.StartStopCommand_003.bVal := FALSE;
                                    5: 
                                        
                                        FB_Bacnet.StartStopCommand_004.bEnWrite := TRUE;
                                        FB_Bacnet.StartStopCommand_004.bVal := FALSE;
                                    6: 
                                        
                                        FB_Bacnet.StartStopCommand_005.bEnWrite := TRUE;
                                        FB_Bacnet.StartStopCommand_005.bVal := FALSE;
                                    7: 
                                        
                                        FB_Bacnet.StartStopCommand_006.bEnWrite := TRUE;
                                        FB_Bacnet.StartStopCommand_006.bVal := FALSE;
                                    8: 
                                        
                                        FB_Bacnet.StartStopCommand_007.bEnWrite := TRUE;
                                        FB_Bacnet.StartStopCommand_007.bVal := FALSE;
                                    9: 
                                        
                                        FB_Bacnet.StartStopCommand_008.bEnWrite := TRUE;
                                        FB_Bacnet.StartStopCommand_008.bVal := FALSE;
                                    10: 
                                        
                                        FB_Bacnet.StartStopCommand_009.bEnWrite := TRUE;
                                        FB_Bacnet.StartStopCommand_009.bVal := FALSE;
                                    11: 
                                        
                                        FB_Bacnet.StartStopCommand_010.bEnWrite := TRUE;
                                        FB_Bacnet.StartStopCommand_010.bVal := FALSE;
                                    12: 
                                        
                                        FB_Bacnet.StartStopCommand_011.bEnWrite := TRUE;
                                        FB_Bacnet.StartStopCommand_011.bVal := FALSE;
                                    13: 
                                        
                                        FB_Bacnet.StartStopCommand_012.bEnWrite := TRUE;
                                        FB_Bacnet.StartStopCommand_012.bVal := FALSE;
                                    14: 
                                        
                                        FB_Bacnet.StartStopCommand_013.bEnWrite := TRUE;
                                        FB_Bacnet.StartStopCommand_013.bVal := FALSE;
                                    15: 
                                        
                                        FB_Bacnet.StartStopCommand_014.bEnWrite := TRUE;
                                        FB_Bacnet.StartStopCommand_014.bVal := FALSE;
                                    16: 
                                        
                                        FB_Bacnet.StartStopCommand_015.bEnWrite := TRUE;
                                        FB_Bacnet.StartStopCommand_015.bVal := FALSE;
                                    17: 
                                        
                                        FB_Bacnet.StartStopCommand_016.bEnWrite := TRUE;
                                        FB_Bacnet.StartStopCommand_016.bVal := FALSE;
                                    18: 
                                        
                                        FB_Bacnet.StartStopCommand_017.bEnWrite := TRUE;
                                        FB_Bacnet.StartStopCommand_017.bVal := FALSE;
                                    19: 
                                        
                                        FB_Bacnet.StartStopCommand_018.bEnWrite := TRUE;
                                        FB_Bacnet.StartStopCommand_018.bVal := FALSE;
                                    20: 
                                        
                                        FB_Bacnet.StartStopCommand_019.bEnWrite := TRUE;
                                        FB_Bacnet.StartStopCommand_019.bVal := FALSE;
                                    21: 
                                        
                                        FB_Bacnet.StartStopCommand_020.bEnWrite := TRUE;
                                        FB_Bacnet.StartStopCommand_020.bVal := FALSE;
                                    22: 
                                        
                                        FB_Bacnet_b.StartStopCommand_225.bEnWrite := TRUE;
                                        FB_Bacnet_b.StartStopCommand_225.bVal := FALSE;
                                END_CASE
                            END_IF
                        END_FOR
                    END_IF
                END_IF
            END_IF
        END_IF

END_FUNCTION_BLOCK

// ---- POUs/FB_Scheduler/FB_Scheduler_F10.TcPOU
FUNCTION_BLOCK FB_Scheduler_F10
    VAR_INPUT
        currH : WORD;
        currM : WORD;
        currD : WORD;
		currDate : WORD;
    END_VAR
    VAR_IN_OUT
        FB_Bacnet : FB_BACnet_DAIKIN_MasterStation_III_No_3;
        FB_Bacnet_b : FB_BACnet_DAIKIN_MasterStation_III_No_2;
    END_VAR
    VAR
        i : INT;
        bUnitTriggered : BOOL := FALSE; // Flag to track execution
        prevMinute : WORD := 0;        // Track previous minute
    END_VAR
    VAR PERSISTENT
        // Scheduler variables
        bEnSchedF10_ : BOOL := FALSE;
        wSchedWDHourStartF10_, wSchedWDMinStartF10_ : WORD;
        wSchedWEHourStartF10_, wSchedWEMinStartF10_ : WORD;
        wSchedWDHourEndF10_, wSchedWDMinEndF10_ : WORD;
        wSchedWEHourEndF10_, wSchedWEMinEndF10_ : WORD;
        // Unit variables
        bUnitF10_ : ARRAY [1..24] OF BOOL;
    END_VAR


// Reset trigger flag at minute change or at the exact scheduled time
IF currM <> prevMinute OR 
   (currH = wSchedWDHourStartF10_ AND currM = wSchedWDMinStartF10_) OR 
   (currH = wSchedWDHourEndF10_ AND currM = wSchedWDMinEndF10_) THEN
    bUnitTriggered := FALSE;
    prevMinute := currM;
END_IF

// Unit Schedule Enable
IF bEnSchedF10_ THEN
    // Weekday schedule
    IF currD >= 1 AND currD <= 5 THEN
        IF (wSchedWDHourStartF10_ <> wSchedWDHourEndF10_ OR wSchedWDMinStartF10_ <> wSchedWDMinEndF10_) THEN
            // Schedule Unit ON
            IF wSchedWDHourStartF10_ = currH AND wSchedWDMinStartF10_ = currM AND NOT bUnitTriggered THEN
                bUnitTriggered := TRUE;
                FOR i := 1 TO 24 DO
                    // Send command unit ON
                    IF bUnitF10_[i] THEN 
                        CASE i OF
                            1: FB_Bacnet.StartStopCommand_064.bEnWrite := TRUE;
                               FB_Bacnet.StartStopCommand_064.bVal := TRUE;
                            2: FB_Bacnet.StartStopCommand_065.bEnWrite := TRUE;
                               FB_Bacnet.StartStopCommand_065.bVal := TRUE;
                            3: FB_Bacnet.StartStopCommand_066.bEnWrite := TRUE;
                               FB_Bacnet.StartStopCommand_066.bVal := TRUE;
                            4: FB_Bacnet.StartStopCommand_067.bEnWrite := TRUE;
                               FB_Bacnet.StartStopCommand_067.bVal := TRUE;
                            5: FB_Bacnet.StartStopCommand_068.bEnWrite := TRUE;
                               FB_Bacnet.StartStopCommand_068.bVal := TRUE;
                            6: FB_Bacnet.StartStopCommand_069.bEnWrite := TRUE;
                               FB_Bacnet.StartStopCommand_069.bVal := TRUE;
                            7: FB_Bacnet.StartStopCommand_070.bEnWrite := TRUE;
                               FB_Bacnet.StartStopCommand_070.bVal := TRUE;
                            8: FB_Bacnet.StartStopCommand_071.bEnWrite := TRUE;
                               FB_Bacnet.StartStopCommand_071.bVal := TRUE;
                            9: FB_Bacnet.StartStopCommand_072.bEnWrite := TRUE;
                               FB_Bacnet.StartStopCommand_072.bVal := TRUE;
                            10: FB_Bacnet.StartStopCommand_073.bEnWrite := TRUE;
                                FB_Bacnet.StartStopCommand_073.bVal := TRUE;
                            11: FB_Bacnet.StartStopCommand_074.bEnWrite := TRUE;
                                FB_Bacnet.StartStopCommand_074.bVal := TRUE;
                            12: FB_Bacnet.StartStopCommand_075.bEnWrite := TRUE;
                                FB_Bacnet.StartStopCommand_075.bVal := TRUE;
                            13: FB_Bacnet.StartStopCommand_076.bEnWrite := TRUE;
                                FB_Bacnet.StartStopCommand_076.bVal := TRUE;
                            14: FB_Bacnet.StartStopCommand_077.bEnWrite := TRUE;
                                FB_Bacnet.StartStopCommand_077.bVal := TRUE;
                            15: FB_Bacnet.StartStopCommand_078.bEnWrite := TRUE;
                                FB_Bacnet.StartStopCommand_078.bVal := TRUE;
                            16: FB_Bacnet.StartStopCommand_079.bEnWrite := TRUE;
                                FB_Bacnet.StartStopCommand_079.bVal := TRUE;
                            17: FB_Bacnet.StartStopCommand_080.bEnWrite := TRUE;
                                FB_Bacnet.StartStopCommand_080.bVal := TRUE;
                            18: FB_Bacnet.StartStopCommand_081.bEnWrite := TRUE;
                                FB_Bacnet.StartStopCommand_081.bVal := TRUE;
                            19: FB_Bacnet.StartStopCommand_082.bEnWrite := TRUE;
                                FB_Bacnet.StartStopCommand_082.bVal := TRUE;
                            20: FB_Bacnet.StartStopCommand_083.bEnWrite := TRUE;
                                FB_Bacnet.StartStopCommand_083.bVal := TRUE;
                            21: FB_Bacnet.StartStopCommand_084.bEnWrite := TRUE;
                                FB_Bacnet.StartStopCommand_084.bVal := TRUE;
                            22: FB_Bacnet.StartStopCommand_112.bEnWrite := TRUE;
                                FB_Bacnet.StartStopCommand_112.bVal := TRUE;
                            23: // FB_Bacnet_b.StartStopCommand_241.bEnWrite := TRUE;
                                // FB_Bacnet_b.StartStopCommand_241.bVal := TRUE;
                            24: FB_Bacnet_b.StartStopCommand_226.bEnWrite := TRUE;
                                FB_Bacnet_b.StartStopCommand_226.bVal := TRUE;
                        END_CASE
                    END_IF
                END_FOR
            END_IF
            // Schedule Unit OFF
            IF wSchedWDHourEndF10_ = currH AND wSchedWDMinEndF10_ = currM AND NOT bUnitTriggered THEN
                bUnitTriggered := TRUE;
                FOR i := 1 TO 24 DO
                    // Send command unit OFF
                    IF bUnitF10_[i] THEN 
                        CASE i OF
                            1: FB_Bacnet.StartStopCommand_064.bEnWrite := TRUE;
                               FB_Bacnet.StartStopCommand_064.bVal := FALSE;
                            2: FB_Bacnet.StartStopCommand_065.bEnWrite := TRUE;
                               FB_Bacnet.StartStopCommand_065.bVal := FALSE;
                            3: FB_Bacnet.StartStopCommand_066.bEnWrite := TRUE;
                               FB_Bacnet.StartStopCommand_066.bVal := FALSE;
                            4: FB_Bacnet.StartStopCommand_067.bEnWrite := TRUE;
                               FB_Bacnet.StartStopCommand_067.bVal := FALSE;
                            5: FB_Bacnet.StartStopCommand_068.bEnWrite := TRUE;
                               FB_Bacnet.StartStopCommand_068.bVal := FALSE;
                            6: FB_Bacnet.StartStopCommand_069.bEnWrite := TRUE;
                               FB_Bacnet.StartStopCommand_069.bVal := FALSE;
                            7: FB_Bacnet.StartStopCommand_070.bEnWrite := TRUE;
                               FB_Bacnet.StartStopCommand_070.bVal := FALSE;
                            8: FB_Bacnet.StartStopCommand_071.bEnWrite := TRUE;
                               FB_Bacnet.StartStopCommand_071.bVal := FALSE;
                            9: FB_Bacnet.StartStopCommand_072.bEnWrite := TRUE;
                               FB_Bacnet.StartStopCommand_072.bVal := FALSE;
                            10: FB_Bacnet.StartStopCommand_073.bEnWrite := TRUE;
                                FB_Bacnet.StartStopCommand_073.bVal := FALSE;
                            11: FB_Bacnet.StartStopCommand_074.bEnWrite := TRUE;
                                FB_Bacnet.StartStopCommand_074.bVal := FALSE;
                            12: FB_Bacnet.StartStopCommand_075.bEnWrite := TRUE;
                                FB_Bacnet.StartStopCommand_075.bVal := FALSE;
                            13: FB_Bacnet.StartStopCommand_076.bEnWrite := TRUE;
                                FB_Bacnet.StartStopCommand_076.bVal := FALSE;
                            14: FB_Bacnet.StartStopCommand_077.bEnWrite := TRUE;
                                FB_Bacnet.StartStopCommand_077.bVal := FALSE;
                            15: FB_Bacnet.StartStopCommand_078.bEnWrite := TRUE;
                                FB_Bacnet.StartStopCommand_078.bVal := FALSE;
                            16: FB_Bacnet.StartStopCommand_079.bEnWrite := TRUE;
                                FB_Bacnet.StartStopCommand_079.bVal := FALSE;
                            17: FB_Bacnet.StartStopCommand_080.bEnWrite := TRUE;
                                FB_Bacnet.StartStopCommand_080.bVal := FALSE;
                            18: FB_Bacnet.StartStopCommand_081.bEnWrite := TRUE;
                                FB_Bacnet.StartStopCommand_081.bVal := FALSE;
                            19: FB_Bacnet.StartStopCommand_082.bEnWrite := TRUE;
                                FB_Bacnet.StartStopCommand_082.bVal := FALSE;
                            20: FB_Bacnet.StartStopCommand_083.bEnWrite := TRUE;
                                FB_Bacnet.StartStopCommand_083.bVal := FALSE;
                            21: FB_Bacnet.StartStopCommand_084.bEnWrite := TRUE;
                                FB_Bacnet.StartStopCommand_084.bVal := FALSE;
                            22: FB_Bacnet.StartStopCommand_112.bEnWrite := TRUE;
                                FB_Bacnet.StartStopCommand_112.bVal := FALSE;
                            23: // FB_Bacnet_b.StartStopCommand_241.bEnWrite := TRUE;
                                // FB_Bacnet_b.StartStopCommand_241.bVal := FALSE;
                            24: FB_Bacnet_b.StartStopCommand_226.bEnWrite := TRUE;
                                FB_Bacnet_b.StartStopCommand_226.bVal := FALSE;
                        END_CASE
                    END_IF
                END_FOR
            END_IF
        END_IF
    END_IF

    // Weekend schedule
    IF currD = 0 OR currD = 6 THEN
        IF (wSchedWEHourStartF10_ <> wSchedWEHourEndF10_ OR wSchedWEMinStartF10_ <> wSchedWEMinEndF10_) THEN
            // Schedule Unit ON
            IF wSchedWEHourStartF10_ = currH AND wSchedWEMinStartF10_ = currM AND NOT bUnitTriggered THEN
                bUnitTriggered := TRUE;
                FOR i := 1 TO 24 DO
                    // Send command unit ON
                    IF bUnitF10_[i] THEN 
                        CASE i OF
                            1: FB_Bacnet.StartStopCommand_064.bEnWrite := TRUE;
                               FB_Bacnet.StartStopCommand_064.bVal := TRUE;
                            2: FB_Bacnet.StartStopCommand_065.bEnWrite := TRUE;
                               FB_Bacnet.StartStopCommand_065.bVal := TRUE;
                            3: FB_Bacnet.StartStopCommand_066.bEnWrite := TRUE;
                               FB_Bacnet.StartStopCommand_066.bVal := TRUE;
                            4: FB_Bacnet.StartStopCommand_067.bEnWrite := TRUE;
                               FB_Bacnet.StartStopCommand_067.bVal := TRUE;
                            5: FB_Bacnet.StartStopCommand_068.bEnWrite := TRUE;
                               FB_Bacnet.StartStopCommand_068.bVal := TRUE;
                            6: FB_Bacnet.StartStopCommand_069.bEnWrite := TRUE;
                               FB_Bacnet.StartStopCommand_069.bVal := TRUE;
                            7: FB_Bacnet.StartStopCommand_070.bEnWrite := TRUE;
                               FB_Bacnet.StartStopCommand_070.bVal := TRUE;
                            8: FB_Bacnet.StartStopCommand_071.bEnWrite := TRUE;
                               FB_Bacnet.StartStopCommand_071.bVal := TRUE;
                            9: FB_Bacnet.StartStopCommand_072.bEnWrite := TRUE;
                               FB_Bacnet.StartStopCommand_072.bVal := TRUE;
                            10: FB_Bacnet.StartStopCommand_073.bEnWrite := TRUE;
                                FB_Bacnet.StartStopCommand_073.bVal := TRUE;
                            11: FB_Bacnet.StartStopCommand_074.bEnWrite := TRUE;
                                FB_Bacnet.StartStopCommand_074.bVal := TRUE;
                            12: FB_Bacnet.StartStopCommand_075.bEnWrite := TRUE;
                                FB_Bacnet.StartStopCommand_075.bVal := TRUE;
                            13: FB_Bacnet.StartStopCommand_076.bEnWrite := TRUE;
                                FB_Bacnet.StartStopCommand_076.bVal := TRUE;
                            14: FB_Bacnet.StartStopCommand_077.bEnWrite := TRUE;
                                FB_Bacnet.StartStopCommand_077.bVal := TRUE;
                            15: FB_Bacnet.StartStopCommand_078.bEnWrite := TRUE;
                                FB_Bacnet.StartStopCommand_078.bVal := TRUE;
                            16: FB_Bacnet.StartStopCommand_079.bEnWrite := TRUE;
                                FB_Bacnet.StartStopCommand_079.bVal := TRUE;
                            17: FB_Bacnet.StartStopCommand_080.bEnWrite := TRUE;
                                FB_Bacnet.StartStopCommand_080.bVal := TRUE;
                            18: FB_Bacnet.StartStopCommand_081.bEnWrite := TRUE;
                                FB_Bacnet.StartStopCommand_081.bVal := TRUE;
                            19: FB_Bacnet.StartStopCommand_082.bEnWrite := TRUE;
                                FB_Bacnet.StartStopCommand_082.bVal := TRUE;
                            20: FB_Bacnet.StartStopCommand_083.bEnWrite := TRUE;
                                FB_Bacnet.StartStopCommand_083.bVal := TRUE;
                            21: FB_Bacnet.StartStopCommand_084.bEnWrite := TRUE;
                                FB_Bacnet.StartStopCommand_084.bVal := TRUE;
                            22: FB_Bacnet.StartStopCommand_112.bEnWrite := TRUE;
                                FB_Bacnet.StartStopCommand_112.bVal := TRUE;
                            23: // FB_Bacnet_b.StartStopCommand_241.bEnWrite := TRUE;
                                // FB_Bacnet_b.StartStopCommand_241.bVal := TRUE;
                            24: FB_Bacnet_b.StartStopCommand_226.bEnWrite := TRUE;
                                FB_Bacnet_b.StartStopCommand_226.bVal := TRUE;
                        END_CASE
                    END_IF
                END_FOR
            END_IF
            // Schedule Unit OFF
            IF wSchedWEHourEndF10_ = currH AND wSchedWEMinEndF10_ = currM AND NOT bUnitTriggered THEN
                bUnitTriggered := TRUE;
                FOR i := 1 TO 24 DO
                    // Send command unit OFF
                    IF bUnitF10_[i] THEN 
                        CASE i OF
                            1: FB_Bacnet.StartStopCommand_064.bEnWrite := TRUE;
                               FB_Bacnet.StartStopCommand_064.bVal := FALSE;
                            2: FB_Bacnet.StartStopCommand_065.bEnWrite := TRUE;
                               FB_Bacnet.StartStopCommand_065.bVal := FALSE;
                            3: FB_Bacnet.StartStopCommand_066.bEnWrite := TRUE;
                               FB_Bacnet.StartStopCommand_066.bVal := FALSE;
                            4: FB_Bacnet.StartStopCommand_067.bEnWrite := TRUE;
                               FB_Bacnet.StartStopCommand_067.bVal := FALSE;
                            5: FB_Bacnet.StartStopCommand_068.bEnWrite := TRUE;
                               FB_Bacnet.StartStopCommand_068.bVal := FALSE;
                            6: FB_Bacnet.StartStopCommand_069.bEnWrite := TRUE;
                               FB_Bacnet.StartStopCommand_069.bVal := FALSE;
                            7: FB_Bacnet.StartStopCommand_070.bEnWrite := TRUE;
                               FB_Bacnet.StartStopCommand_070.bVal := FALSE;
                            8: FB_Bacnet.StartStopCommand_071.bEnWrite := TRUE;
                               FB_Bacnet.StartStopCommand_071.bVal := FALSE;
                            9: FB_Bacnet.StartStopCommand_072.bEnWrite := TRUE;
                               FB_Bacnet.StartStopCommand_072.bVal := FALSE;
                            10: FB_Bacnet.StartStopCommand_073.bEnWrite := TRUE;
                                FB_Bacnet.StartStopCommand_073.bVal := FALSE;
                            11: FB_Bacnet.StartStopCommand_074.bEnWrite := TRUE;
                                FB_Bacnet.StartStopCommand_074.bVal := FALSE;
                            12: FB_Bacnet.StartStopCommand_075.bEnWrite := TRUE;
                                FB_Bacnet.StartStopCommand_075.bVal := FALSE;
                            13: FB_Bacnet.StartStopCommand_076.bEnWrite := TRUE;
                                FB_Bacnet.StartStopCommand_076.bVal := FALSE;
                            14: FB_Bacnet.StartStopCommand_077.bEnWrite := TRUE;
                                FB_Bacnet.StartStopCommand_077.bVal := FALSE;
                            15: FB_Bacnet.StartStopCommand_078.bEnWrite := TRUE;
                                FB_Bacnet.StartStopCommand_078.bVal := FALSE;
                            16: FB_Bacnet.StartStopCommand_079.bEnWrite := TRUE;
                                FB_Bacnet.StartStopCommand_079.bVal := FALSE;
                            17: FB_Bacnet.StartStopCommand_080.bEnWrite := TRUE;
                                FB_Bacnet.StartStopCommand_080.bVal := FALSE;
                            18: FB_Bacnet.StartStopCommand_081.bEnWrite := TRUE;
                                FB_Bacnet.StartStopCommand_081.bVal := FALSE;
                            19: FB_Bacnet.StartStopCommand_082.bEnWrite := TRUE;
                                FB_Bacnet.StartStopCommand_082.bVal := FALSE;
                            20: FB_Bacnet.StartStopCommand_083.bEnWrite := TRUE;
                                FB_Bacnet.StartStopCommand_083.bVal := FALSE;
                            21: FB_Bacnet.StartStopCommand_084.bEnWrite := TRUE;
                                FB_Bacnet.StartStopCommand_084.bVal := FALSE;
                            22: FB_Bacnet.StartStopCommand_112.bEnWrite := TRUE;
                                FB_Bacnet.StartStopCommand_112.bVal := FALSE;
                            23: // FB_Bacnet_b.StartStopCommand_241.bEnWrite := TRUE;
                                // FB_Bacnet_b.StartStopCommand_241.bVal := FALSE;
                            24: FB_Bacnet_b.StartStopCommand_226.bEnWrite := TRUE;
                                FB_Bacnet_b.StartStopCommand_226.bVal := FALSE;
                        END_CASE
                    END_IF
                END_FOR
            END_IF
        END_IF
    END_IF
END_IF

END_FUNCTION_BLOCK

// ---- POUs/FB_Scheduler/FB_Scheduler_F11.TcPOU

      FUNCTION_BLOCK FB_Scheduler_F11
      VAR_INPUT
          currH : WORD;
          currM : WORD;
          currD : WORD;
      END_VAR
      VAR_IN_OUT
          FB_Bacnet : FB_BACnet_DAIKIN_MasterStation_III_No_3;
          FB_Bacnet_b : FB_BACnet_DAIKIN_MasterStation_III_No_2;
      END_VAR
      VAR
          i : INT;
          bUnitTriggered : BOOL := FALSE; // New flag to track execution
          prevMinute : WORD := 0;        // New variable to track the previous minute
      END_VAR
      VAR PERSISTENT
          //scheduler var
          bEnSchedF11_ : BOOL := FALSE;
          wSchedWDHourStartF11_ : WORD; 
          wSchedWDMinStartF11_ : WORD; 
          wSchedWEHourStartF11_ : WORD; 
          wSchedWEMinStartF11_ : WORD;
          wSchedWDHourEndF11_ : WORD;
          wSchedWDMinEndF11_ : WORD;
          wSchedWEHourEndF11_ : WORD;
          wSchedWEMinEndF11_ : WORD;
          //unit var
          bUnitF11_ : ARRAY [1..22] OF BOOL;
      END_VAR


        // Reset trigger flag at minute change or at the exact scheduled time
        IF currM <> prevMinute OR 
           (currH = wSchedWDHourStartF11_ AND currM = wSchedWDMinStartF11_) OR 
           (currH = wSchedWDHourEndF11_ AND currM = wSchedWDMinEndF11_) THEN
            bUnitTriggered := FALSE;
            prevMinute := currM;
        END_IF

        // Unit Schedule Enable
        IF bEnSchedF11_ THEN
            // Weekday schedule
            IF currD >= 1 AND currD <= 5 THEN
                IF (wSchedWDHourStartF11_ <> wSchedWDHourEndF11_ OR wSchedWDMinStartF11_ <> wSchedWDMinEndF11_) THEN
                    // Schedule Unit ON
                    IF wSchedWDHourStartF11_ = currH AND wSchedWDMinStartF11_ = currM AND NOT bUnitTriggered THEN
                        bUnitTriggered := TRUE;
                        FOR i := 1 TO 22 DO
                            // Send command unit ON
                            IF bUnitF11_[i] THEN 
                                CASE i OF
                                    1: 
                                        //
                                        //FB_Bacnet.StartStopCommand_128.bEnWrite := TRUE;
                                        //FB_Bacnet.StartStopCommand_128.bVal := TRUE;
                                    2: 
                                        //
                                        //FB_Bacnet.StartStopCommand_129.bEnWrite := TRUE;
                                        //FB_Bacnet.StartStopCommand_129.bVal := TRUE;
                                    3: 
                                        (*
                                        FB_Bacnet.StartStopCommand_130.bEnWrite := TRUE;
                                        FB_Bacnet.StartStopCommand_130.bVal := TRUE;*)
                                    4: 
                                        //
                                        //FB_Bacnet.StartStopCommand_131.bEnWrite := TRUE;
                                        //FB_Bacnet.StartStopCommand_131.bVal := TRUE;
                                    5: 
                                        (*
                                        FB_Bacnet.StartStopCommand_132.bEnWrite := TRUE;
                                        FB_Bacnet.StartStopCommand_132.bVal := TRUE;*)
                                    6: 
                                        //
                                        //FB_Bacnet.StartStopCommand_133.bEnWrite := TRUE;
                                        //FB_Bacnet.StartStopCommand_133.bVal := TRUE;
                                    7: 
                                        //
                                        //FB_Bacnet.StartStopCommand_134.bEnWrite := TRUE;
                                        //FB_Bacnet.StartStopCommand_134.bVal := TRUE;
                                    8: 
                                        //
                                        //FB_Bacnet.StartStopCommand_135.bEnWrite := TRUE;
                                        //FB_Bacnet.StartStopCommand_135.bVal := TRUE;
                                    9: 
                                        //
                                        //FB_Bacnet.StartStopCommand_136.bEnWrite := TRUE;
                                        //FB_Bacnet.StartStopCommand_136.bVal := TRUE;
                                    10: 
                                        //
                                        //FB_Bacnet.StartStopCommand_137.bEnWrite := TRUE;
                                        //FB_Bacnet.StartStopCommand_137.bVal := TRUE;
                                    11: 
                                        //
                                        //FB_Bacnet.StartStopCommand_138.bEnWrite := TRUE;
                                        //FB_Bacnet.StartStopCommand_138.bVal := TRUE;
                                    12: 
                                        //
                                        //FB_Bacnet.StartStopCommand_139.bEnWrite := TRUE;
                                        //FB_Bacnet.StartStopCommand_139.bVal := TRUE;
                                    13: 
                                        //
                                        //FB_Bacnet.StartStopCommand_140.bEnWrite := TRUE;
                                        //FB_Bacnet.StartStopCommand_140.bVal := TRUE;
                                    14: 
                                        //
                                        //FB_Bacnet.StartStopCommand_141.bEnWrite := TRUE;
                                        //FB_Bacnet.StartStopCommand_141.bVal := TRUE;
                                    15: 
                                        (*
                                        FB_Bacnet.StartStopCommand_142.bEnWrite := TRUE;
                                        FB_Bacnet.StartStopCommand_142.bVal := TRUE;*)
                                    16: 
                                        (*
                                        FB_Bacnet.StartStopCommand_143.bEnWrite := TRUE;
                                        FB_Bacnet.StartStopCommand_143.bVal := TRUE;*)
                                    17: 
                                        
                                        FB_Bacnet.StartStopCommand_144.bEnWrite := TRUE;
                                        FB_Bacnet.StartStopCommand_144.bVal := TRUE;
                                    18: 
                                        //
                                        //FB_Bacnet.StartStopCommand_145.bEnWrite := TRUE;
                                        //FB_Bacnet.StartStopCommand_145.bVal := TRUE;
                                    19: 
                                        //
                                        //FB_Bacnet.StartStopCommand_146.bEnWrite := TRUE;
                                        //FB_Bacnet.StartStopCommand_146.bVal := TRUE;
                                    20: 
                                        //
                                        //FB_Bacnet.StartStopCommand_147.bEnWrite := TRUE;
                                        //FB_Bacnet.StartStopCommand_147.bVal := TRUE;
                                    21: 
                                        //
                                        //FB_Bacnet.StartStopCommand_148.bEnWrite := TRUE;
                                        //FB_Bacnet.StartStopCommand_148.bVal := TRUE;
                                    22: 
                                        
                                        FB_Bacnet_b.StartStopCommand_227.bEnWrite := TRUE;
                                        FB_Bacnet_b.StartStopCommand_227.bVal := TRUE;
                                END_CASE
                            END_IF
                        END_FOR
                    END_IF
                    // Schedule Unit OFF
                    IF wSchedWDHourEndF11_ = currH AND wSchedWDMinEndF11_ = currM AND NOT bUnitTriggered THEN
                        bUnitTriggered := TRUE;
                        FOR i := 1 TO 22 DO
                            // Send command unit OFF
                            IF bUnitF11_[i] THEN 
                                CASE i OF
                                    1: 
                                        //
                                        //FB_Bacnet.StartStopCommand_128.bEnWrite := TRUE;
                                        //FB_Bacnet.StartStopCommand_128.bVal := FALSE;
                                    2: 
                                        //
                                        //FB_Bacnet.StartStopCommand_129.bEnWrite := TRUE;
                                        //FB_Bacnet.StartStopCommand_129.bVal := FALSE;
                                    3: 
                                        //
                                        //FB_Bacnet.StartStopCommand_130.bEnWrite := TRUE;
                                        //FB_Bacnet.StartStopCommand_130.bVal := FALSE;
                                    4: 
                                        //
                                        //FB_Bacnet.StartStopCommand_131.bEnWrite := TRUE;
                                        //FB_Bacnet.StartStopCommand_131.bVal := FALSE;
                                    5: 
                                        //
                                        //FB_Bacnet.StartStopCommand_132.bEnWrite := TRUE;
                                        //FB_Bacnet.StartStopCommand_132.bVal := FALSE;
                                    6: 
                                        //
                                        //FB_Bacnet.StartStopCommand_133.bEnWrite := TRUE;
                                        //FB_Bacnet.StartStopCommand_133.bVal := FALSE;
                                    7: 
                                        //
                                        //FB_Bacnet.StartStopCommand_134.bEnWrite := TRUE;
                                        //FB_Bacnet.StartStopCommand_134.bVal := FALSE;
                                    8: 
                                        //
                                        //FB_Bacnet.StartStopCommand_135.bEnWrite := TRUE;
                                        //FB_Bacnet.StartStopCommand_135.bVal := FALSE;
                                    9: 
                                        //
                                        //FB_Bacnet.StartStopCommand_136.bEnWrite := TRUE;
                                        //FB_Bacnet.StartStopCommand_136.bVal := FALSE;
                                    10: 
                                        //
                                        //FB_Bacnet.StartStopCommand_137.bEnWrite := TRUE;
                                        //FB_Bacnet.StartStopCommand_137.bVal := FALSE;
                                    11: 
                                        //
                                        //FB_Bacnet.StartStopCommand_138.bEnWrite := TRUE;
                                        //FB_Bacnet.StartStopCommand_138.bVal := FALSE;
                                    12: 
                                        //
                                        //FB_Bacnet.StartStopCommand_139.bEnWrite := TRUE;
                                        //FB_Bacnet.StartStopCommand_139.bVal := FALSE;
                                    13: 
                                        //
                                        //FB_Bacnet.StartStopCommand_140.bEnWrite := TRUE;
                                        //FB_Bacnet.StartStopCommand_140.bVal := FALSE;
                                    14: 
                                        //
                                        //FB_Bacnet.StartStopCommand_141.bEnWrite := TRUE;
                                        //FB_Bacnet.StartStopCommand_141.bVal := FALSE;
                                    15: 
                                        //
                                        //FB_Bacnet.StartStopCommand_142.bEnWrite := TRUE;
                                        //FB_Bacnet.StartStopCommand_142.bVal := FALSE;
                                    16: 
                                        //
                                        //FB_Bacnet.StartStopCommand_143.bEnWrite := TRUE;
                                        //FB_Bacnet.StartStopCommand_143.bVal := FALSE;
                                    17: 
                                        //
                                        //FB_Bacnet.StartStopCommand_144.bEnWrite := TRUE;
                                        //FB_Bacnet.StartStopCommand_144.bVal := FALSE;
                                    18: 
                                        //
                                        //FB_Bacnet.StartStopCommand_145.bEnWrite := TRUE;
                                        //FB_Bacnet.StartStopCommand_145.bVal := FALSE;
                                    19: 
                                        //
                                        //FB_Bacnet.StartStopCommand_146.bEnWrite := TRUE;
                                        //FB_Bacnet.StartStopCommand_146.bVal := FALSE;
                                    20: 
                                        //
                                        //FB_Bacnet.StartStopCommand_147.bEnWrite := TRUE;
                                        //FB_Bacnet.StartStopCommand_147.bVal := FALSE;
                                    21: 
                                        //
                                        //FB_Bacnet.StartStopCommand_148.bEnWrite := TRUE;
                                        //FB_Bacnet.StartStopCommand_148.bVal := FALSE;
                                    22: 
                                        
                                        FB_Bacnet_b.StartStopCommand_227.bEnWrite := TRUE;
                                        FB_Bacnet_b.StartStopCommand_227.bVal := FALSE;
                                END_CASE
                            END_IF
                        END_FOR
                    END_IF
                END_IF
            END_IF

